KUKA KRL program: Outputs.src

&ACCESS RV
DEF Outputs ( )

   CONTINUE
   OUT_RobotUnknowPos = boRobotUnknowPos

 ;;  boButtonPanel = biStartProgram

  ;; CONTINUE
   ;;OUT_ButtonPanel = boButtonPanel

END
